Fanuc KAREL source: port_LDO.kl

PROGRAM TP
%NOLOCKGROUP
VAR
 x: BOOLEAN
BEGIN
 x = LDO[3]
END TP
